FUNCTION_BLOCK FB_EventFMZ2
VAR_INPUT
	FB_Bacnet : FB_BACnet_DAIKIN_MasterStation_III_No_1;
END_VAR
VAR_OUTPUT
END_VAR
VAR
	fbMsg : FB_TcMessage;
	aUnits : ARRAY[1..8] OF AC_Unit_Status;
	stUnit   : AC_Unit_Status;
	i: INT;
	sMsgText: STRING;
	triggerTest : BOOL;
END_VAR
VAR RETAIN
	aPrevState : ARRAY[1..8] OF BOOL := [FALSE(*8*)];
END_VAR


aUnits[1].bPresVal := FB_Bacnet.StartStopStatus_096.bPresVal;
aUnits[1].sUnitName := 'FMZ-PC-1 (3-00)';
aUnits[2].bPresVal := FB_Bacnet.StartStopStatus_097.bPresVal;
aUnits[2].sUnitName := 'FMZ-PC-2 (3-01)';
aUnits[3].bPresVal := FB_Bacnet.StartStopStatus_098.bPresVal;
aUnits[3].sUnitName := 'FMZ-PC-3 (3-02)';
aUnits[4].bPresVal := FB_Bacnet.StartStopStatus_099.bPresVal;
aUnits[4].sUnitName := 'FMZ-PC-4 (3-03)';
aUnits[5].bPresVal := FB_Bacnet.StartStopStatus_100.bPresVal;
aUnits[5].sUnitName := 'FMZ-PC-5 (3-04)';
aUnits[6].bPresVal := FB_Bacnet.StartStopStatus_101.bPresVal;
aUnits[6].sUnitName := 'FMZ-PC-6 (3-05)';
aUnits[7].bPresVal := FB_Bacnet.StartStopStatus_102.bPresVal;
aUnits[7].sUnitName := 'FMZ-PC-7 (3-06)';
aUnits[8].bPresVal := FB_Bacnet.StartStopStatus_103.bPresVal;
aUnits[8].sUnitName := 'FMZ-PC-8 (3-07)';

FOR i := 1 TO 8 DO
	stUnit := aUnits[i]; // extract the structure instance
    IF aUnits[i].bPresVal <> aPrevState[i] THEN
        IF aUnits[i].bPresVal THEN
            sMsgText := CONCAT(stUnit.sUnitName, ' is Turned ON');
        ELSE
            sMsgText := CONCAT(stUnit.sUnitName, ' is Turned OFF');
        END_IF
		fbMsg.CreateEx(TC_EVENTS.UnitPowerStatus.EventPowerStatus, 0);
		fbMsg.ipArguments.AddString(sMsgText);
		fbMsg.Send(0);
		
        // Update previous state
        aPrevState[i] := aUnits[i].bPresVal;
    END_IF
END_FOR

END_FUNCTION_BLOCK

(* stored: Version 1.1.0.1, ProductVersion 3.1.4024.14
   POU FB_EventFMZ2: Id {c95ee243-04a3-4807-ae16-2a2489f80775}, SpecialFunc None *)
